{attribute 'GeneratedUsingTerminal: EL3001-0000-0016'}
{attribute addProperty BoxType "EL3001-0000-0016"}
{attribute addProperty Id "UnderrangeAT %I*BOOL1OverrangeAT %I*BOOL1Limit_xAT %I*ARRAY[0..1] OF BYTE2ErrorAT %I*BOOL1TxPDO_StateAT %I*BOOL1TxPDO_ToggleAT %I*BOOL1ValueAT %I*INT2"}
{attribute addProperty CRC "1583108878"}
{attribute addProperty Size "9"}
TYPE AI_Standard_EA9DF21E :
STRUCT
	{attribute addProperty Name "Underrange"}
	Underrange AT %I* : BOOL;
	{attribute addProperty Name "Overrange"}
	Overrange AT %I* : BOOL;
	{attribute addProperty Name "Limit"}
	Limit_x AT %I* : ARRAY[0..1] OF BYTE;
	{attribute addProperty Name "Error"}
	Error AT %I* : BOOL;
	{attribute addProperty Name "TxPDO_State"}
	TxPDO_State AT %I* : BOOL;
	{attribute addProperty Name "TxPDO_Toggle"}
	TxPDO_Toggle AT %I* : BOOL;
	{attribute addProperty Name "Value"}
	Value AT %I* : INT;
END_STRUCT
END_TYPE

(* stored: Version 1.2.0.0, ProductVersion 3.1.4024.9
   DUT AI_Standard_EA9DF21E: Id {eaefe32f-2a10-4a2a-b562-18f805842c02} *)
